(* Schneider Machine Expert - Basic project program_, file version 2.7.0.0 *)
(* ProjectInformations: Name=New project *)

HARDWARE
  Cpu 0: TM200CE40T
  EthernetConfiguration: NetworkName=M200, IpAllocationMode=FixedAddress, IpAddress=192.168.1.15, SubnetMask=255.255.255.0
  SerialLineConfiguration: Baud=Baud9600, Parity=ParityNone, DataBits=DataBits8, StopBits=StopBits1, PhysicalMedium=PhysicalMediumRs485, TransmissionMode=TransmissionModeModbusRtu, SlaveId=1, Addressing=SlaveAddressing
  MastTask: UsePeriodScanMode=false, PeriodScan=100
  FastTask: Period=255
  CpuBehavior: StartingMode=StartAsPreviousState, AutoSaveRamOnEeprom=true, WatchdogPeriod=250

SYMBOLS  (address, symbol, comment, settings)
  %M0       SERIAL_PARSING
  %M5       RESET_COUNTER
  %S5       SB_TB100MS  "Time base of 100 ms generated by an internal clock"
  %MW4      NILAI_COUNTER
  %MW7      REAL_VALUE_COUNTER
  %MF10     ROTARY_SPEED
  %MF31     EXHAUST_GAS_TEMP
  %MF34     MAIN_BEARING_TEMP
  %TM0        [Preset=1, Base=OneSecond]
  %READ_VAR0   [Link(Value(FBComLinkParameterEnums=SerialLine1)), RemoteDeviceId(Value(int=1)), Timeout(Value(int=100)), ObjType(Value(FBComObjTypeParameterEnums=MW)), FirstObj(Value(int=0)), Quantity(Value(int=5)), IndexData(Value(int=250))]
  %I0.1     INPUT_PROXIMITY
  %Q0.0     LAMP_NORMAL
  %Q0.1     LAMP_WARNING
  %Q0.2     LAMP_DANGER

POU Sensor Proximity
  (* SectionNumber=1 *)

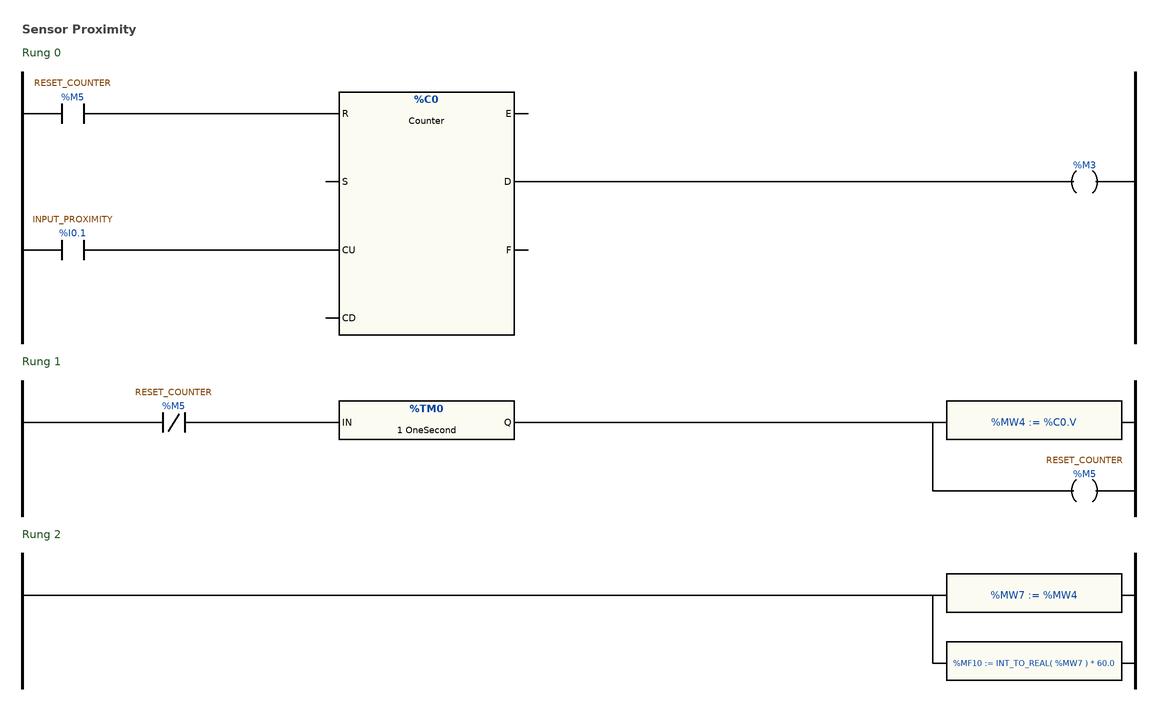

// Rung 0
  BLK %C0
  LD %M5                  (* RESET_COUNTER *)
  R
  LD %I0.1                (* INPUT_PROXIMITY *)
  CU
  OUT_BLK
  LD D
  ST %M3
  END_BLK
  // as ST:
  //   %C0(R := RESET_COUNTER, CU := INPUT_PROXIMITY);
  //   %M3 := %C0.D;

// Rung 1
  BLK %TM0
  LDN %M5                 (* RESET_COUNTER *)
  IN
  OUT_BLK
  LD Q
  [ %MW4 := %C0.V ]       (* NILAI_COUNTER *)
  ST %M5                  (* RESET_COUNTER *)
  END_BLK
  // as ST:
  //   %TM0(IN := NOT RESET_COUNTER);
  //   IF %TM0.Q THEN NILAI_COUNTER := %C0.V; END_IF;
  //   RESET_COUNTER := %TM0.Q;

// Rung 2
  LD 1
  [ %MW7 := %MW4 ]        (* REAL_VALUE_COUNTER, NILAI_COUNTER *)
  [%MF10 := INT_TO_REAL( %MW7 ) * 60.0](* ROTARY_SPEED, REAL_VALUE_COUNTER *)
  // as ST:
  //   REAL_VALUE_COUNTER := NILAI_COUNTER;
  //   ROTARY_SPEED := INT_TO_REAL( REAL_VALUE_COUNTER ) * 60.0;

POU Serial Data
  (* SectionNumber=2 *)

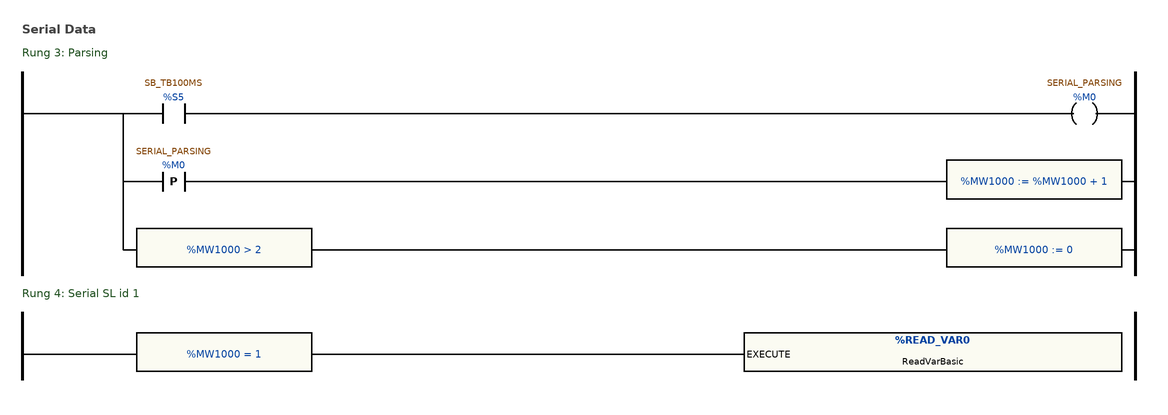

// Rung 3: Parsing
  LD 1
  MPS
  AND %S5                 (* SB_TB100MS *)
  ST %M0                  (* SERIAL_PARSING *)
  MRD
  ANDR %M0                (* SERIAL_PARSING *)
  [ %MW1000 := %MW1000 + 1 ]
  MPP
  AND [ %MW1000 > 2 ]
  [ %MW1000 := 0 ]
  // as ST:
  //   SERIAL_PARSING := SB_TB100MS;
  //   IF RISING(SERIAL_PARSING) THEN %MW1000 := %MW1000 + 1; END_IF;
  //   IF %MW1000 > 2 THEN %MW1000 := 0; END_IF;

// Rung 4: Serial SL id 1
  BLK %READ_VAR0
  LD 1
  AND [ %MW1000 = 1 ]
  EXECUTE
  END_BLK
  // as ST:
  //   %READ_VAR0(EXECUTE := %MW1000 = 1);

POU Temp Data
  (* SectionNumber=3 *)

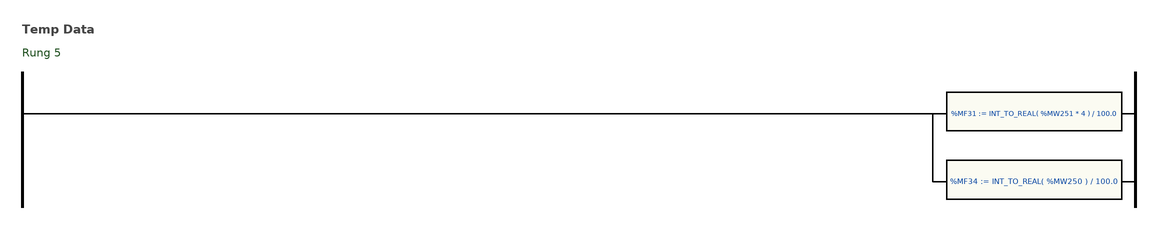

// Rung 5
  LD 1
  [%MF31 := INT_TO_REAL( %MW251 * 4 ) / 100.0](* EXHAUST_GAS_TEMP *)
  [%MF34 := INT_TO_REAL( %MW250 ) / 100.0](* MAIN_BEARING_TEMP *)
  // as ST:
  //   EXHAUST_GAS_TEMP := INT_TO_REAL( %MW251 * 4 ) / 100.0;
  //   MAIN_BEARING_TEMP := INT_TO_REAL( %MW250 ) / 100.0;

POU Indikator System
  (* SectionNumber=4 *)

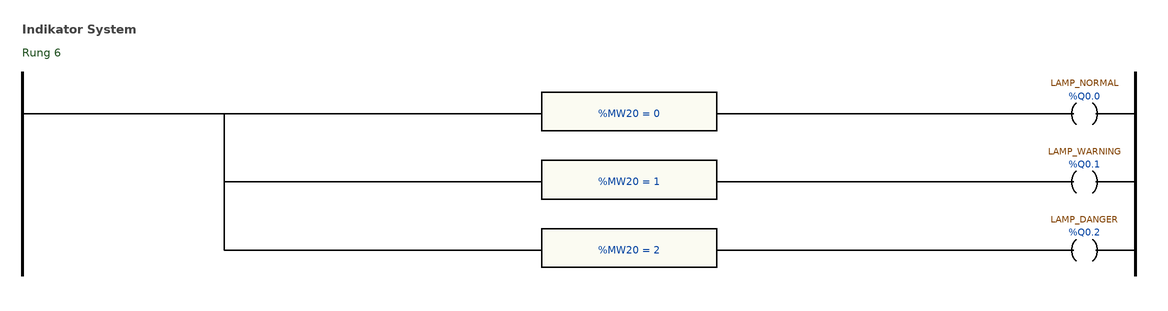

// Rung 6
  LD 1
  MPS
  AND [ %MW20 = 0 ]
  ST %Q0.0                (* LAMP_NORMAL *)
  MRD
  AND [ %MW20 = 1 ]
  ST %Q0.1                (* LAMP_WARNING *)
  MPP
  AND [ %MW20 = 2 ]
  ST %Q0.2                (* LAMP_DANGER *)
  // as ST:
  //   LAMP_NORMAL := %MW20 = 0;
  //   LAMP_WARNING := %MW20 = 1;
  //   LAMP_DANGER := %MW20 = 2;
